(* IEC 61131-3 sources: IRIS-Project/LASAL CONTROL SOFTWARE/LasalProject_2025_09_12/Class/Mode_selector_class, 1 file *)

(* ---- Mode_selector_class.st ---- *)
(*!
<Class
	Name               = "Mode_selector_class"
	Revision           = "0.0"
	RealtimeTask       = "false"
	DefRealtime        = "100 ms"
	CyclicTask         = "true"
	DefCyclictime      = "100 ms"
	BackgroundTask     = "false"
	DefBackground      = "100 ms"
	Sigmatek           = "false"
	OSInterface        = "false"
	HighPriority       = "false"
	Automatic          = "false"
	UpdateMode         = "Prescan"
	SharedCommandTable = "true"
	Objectsize         = "(836,120)">
	<Channels>
		<Server Name="ClassSvr" Visualized="false" Initialize="false" WriteProtected="true" Retentive="false"/>
		<Server Name="Selector" Visualized="false" Initialize="false" WriteProtected="false" Retentive="false"/>
		<Client Name="To_Manager_manual_Motor" Required="true" Internal="false"/>
		<Client Name="To_Manager_motori" Required="true" Internal="false"/>
	</Channels>
</Class>
*)
Mode_selector_class : CLASS
	TYPE
	  T_Selector :  //! <Type Public="true" Name="T_Selector"/>
	  (
	    Automatic:=0,
	    Manual:=1,
	    Idle
	  )$UDINT;
	END_TYPE
  //Servers:
	ClassSvr 	: SvrChCmd_DINT;
	Selector 	: SvrCh_T_Selector_PTofCls_Mode_selector_class;
  //Clients:
	To_Manager_motori 	: CltCh_DINT;
	To_Manager_manual_Motor 	: CltCh_DINT;
  //Variables:
		v_Selector 	: T_Selector;
  //Functions:

	FUNCTION VIRTUAL GLOBAL CyWork
		VAR_INPUT
			EAX 	: UDINT;
		END_VAR
		VAR_OUTPUT
			state (EAX) 	: UDINT;
		END_VAR;

	FUNCTION VIRTUAL GLOBAL Selector::Read
		VAR_OUTPUT
			output (EAX) 	: Mode_selector_class::T_Selector;
		END_VAR;
  //Tables:
	FUNCTION @STD
		VAR_OUTPUT
			ret_code	: CONFSTATES;
		END_VAR;
	FUNCTION GLOBAL TAB @CT_;
END_CLASS;

FUNCTION VIRTUAL GLOBAL Mode_selector_class::Selector::Read
	VAR_OUTPUT
		output (EAX) 	: Mode_selector_class::T_Selector;
	END_VAR

	output := Selector;

END_FUNCTION

FUNCTION VIRTUAL GLOBAL Mode_selector_class::CyWork
	VAR_INPUT
		EAX 	: UDINT;
	END_VAR
	VAR_OUTPUT
		state (EAX) 	: UDINT;
	END_VAR

  v_Selector:=Selector.Read();

  case v_Selector of

    Automatic:
      To_Manager_motori.Write(input:=0);
      To_Manager_manual_Motor.Write(input:=0);

    Manual:
      To_Manager_motori.Write(input:=1);
      To_Manager_manual_Motor.Write(input:=1);

    Idle:

  end_case;

	state := READY;

END_FUNCTION
